// TIA Portal V18 export
VAR_GLOBAL   // PLC tag table "MemoryType"
   "PBB Off Mode Memo" AT %M200.0 : Bool;
   "PBB On Mode Memo" AT %M200.1 : Bool;
   "PBB Auto Mode Memo" AT %M200.2 : Bool;
   "Emergency Stop Button Pressed Memo" AT %M200.3 : Bool;
   "Tunnel FW Em Stop LS M Memo" AT %M200.4 : Bool;
   "Tunnel BW Em Stop LS M Memo" AT %M200.5 : Bool;
   "Start M Memo" AT %M200.6 : Bool;
   "Fuse Problem Major Memo" AT %M200.7 : Bool;
   "AutoLeveller Fault Memo" AT %M201.0 : Bool;
   "AutoLeveller Up Over Work Memo" AT %M201.1 : Bool;
   "AutoLeveller Down Over Work Memo" AT %M201.2 : Bool;
   "Driver Error Left Memo" AT %M201.3 : Bool;
   "Driver Error Right Memo" AT %M201.4 : Bool;
   "Wheel Drivers Fault Memo" AT %M201.5 : Bool;
   "SafetyShoe Siren&Info Memo" AT %M201.6 : Bool;
   "SafetyBarrier Activated Memo" AT %M201.7 : Bool;
   "Service GPU Active Memo" AT %M202.0 : Bool;
   "Fault Occurred Major Memo" AT %M202.1 : Bool;
   "Cabin Motor Driver Fault Memo" AT %M202.2 : Bool;
   "Fault Occured Minor Memo" AT %M202.3 : Bool;
   "OK Memo" AT %M202.4 : Bool;
   "FW L1 Memo" AT %M202.5 : Bool;
   "FW L2 Memo" AT %M202.6 : Bool;
   "FW L3 Memo" AT %M202.7 : Bool;
   "BW L1 Memo" AT %M203.0 : Bool;
   "BW L2 Memo" AT %M203.1 : Bool;
   "BW L3 Memo" AT %M203.2 : Bool;
   "LFT L1 Memo" AT %M203.3 : Bool;
   "LFT L2 Memo" AT %M203.4 : Bool;
   "LFT L3 Memo" AT %M203.5 : Bool;
   "RGHT L1 Memo" AT %M203.6 : Bool;
   "RGHT L2 Memo" AT %M203.7 : Bool;
   "RGHT L3 Memo" AT %M204.0 : Bool;
   "JS Mid M Memo" AT %M204.1 : Bool;
   "SafetyShoe Activated Memo" AT %M204.2 : Bool;
   "AutoLeveller Up Memo" AT %M204.3 : Bool;
   "AutoLeveller Down Memo" AT %M204.4 : Bool;
   "Down Stop Object Limit Memo" AT %M204.6 : Bool;
   "SafetyShoe Long Press Memo" AT %M204.7 : Bool;
   "SS Cable Problem Memo" AT %M205.0 : Bool;
   "AutoSafety Cross Memo" AT %M205.1 : Bool;
   "AutoLeveller FW Memo" AT %M205.2 : Bool;
   "AutoLeveller BW Memo" AT %M205.3 : Bool;
   "Autoleveler temp count Memo" AT %M205.4 : Bool;
   "Service PCA Active Memo" AT %M205.5 : Bool;
   "Service Hose Active Memo" AT %M205.6 : Bool;
   "Fuse Problem Minor Memo" AT %M205.7 : Bool;
   "Wire Up Stop PBB Memo" AT %M206.0 : Bool;
   "Slope Stop Up Memo" AT %M206.1 : Bool;
   "Wire Up Stop PBB Limit All Memo" AT %M206.2 : Bool;
   "Wire Down Stop PBB Memo" AT %M206.3 : Bool;
   "Slope Stop Down Memo" AT %M206.4 : Bool;
   "Down Stop Object Memo" AT %M206.5 : Bool;
   "Down Stop PBB All Memo" AT %M206.6 : Bool;
   "Slope Slow Down Memo" AT %M206.7 : Bool;
   "Slope Slow Up Memo" AT %M207.0 : Bool;
   "Slope Slow ALL Memo" AT %M207.1 : Bool;
   "Slow Activated Memo" AT %M207.2 : Bool;
   "Drive Slow Limit All Memo" AT %M207.3 : Bool;
   "FW Slow Limit All Memo" AT %M207.4 : Bool;
   "BW Slow Limit All Memo" AT %M207.5 : Bool;
   "FW M Memo" AT %M207.6 : Bool;
   "BW M Memo" AT %M207.7 : Bool;
   "FW-LFT Memo" AT %M208.0 : Bool;
   "FW-RGHT Memo" AT %M208.1 : Bool;
   "BW-LFT Memo" AT %M208.2 : Bool;
   "BW-RGHT Memo" AT %M208.3 : Bool;
   "Cross M Memo" AT %M208.4 : Bool;
   "FW Stop All Memo" AT %M208.5 : Bool;
   "BW Stop All Memo" AT %M208.6 : Bool;
   "LFT Stop All Memo" AT %M208.7 : Bool;
   "RGHT Stop All Memo" AT %M209.0 : Bool;
   "FW Allowed Memo" AT %M209.1 : Bool;
   "BW Allowed Memo" AT %M209.2 : Bool;
   "LFT Allowed Memo" AT %M209.3 : Bool;
   "RGHT Allowed Memo" AT %M209.4 : Bool;
   "FW-LFT Allowed Memo" AT %M209.5 : Bool;
   "FW-RGHT Allowed Memo" AT %M209.6 : Bool;
   "BW-LFT Allowed Memo" AT %M209.7 : Bool;
   "BW-RGHT Allowed Memo" AT %M210.0 : Bool;
   "Drive Angle Stop Left Memo" AT %M210.1 : Bool;
   "Drive LSW Left Stop Memo" AT %M210.2 : Bool;
   "Drive Angle Stop Right Memo" AT %M210.3 : Bool;
   "Drive LSW Right Stop Memo" AT %M210.4 : Bool;
   "Drive Slow Left Limit Memo" AT %M210.5 : Bool;
   "Drive Slow Right Limit Memo" AT %M210.6 : Bool;
   "Rotunda FW Stop LFT Memo" AT %M210.7 : Bool;
   "Rotunda BW Stop LFT Memo" AT %M211.0 : Bool;
   "Rotunda FW Stop RGHT Memo" AT %M211.1 : Bool;
   "Rotunda BW Stop RGHT Memo" AT %M211.2 : Bool;
   "Rotunda FW Stop All Memo" AT %M211.3 : Bool;
   "Rotunda BW Stop All Memo" AT %M211.4 : Bool;
   "Tunnel Laser FW Slow Limit Memo" AT %M211.5 : Bool;
   "Tunnel LSW FW Slow Memo" AT %M211.6 : Bool;
   "PhotoCell Slow Limit Memo" AT %M211.7 : Bool;
   "UltraSonic Slow Limit Memo" AT %M212.0 : Bool;
   "AirCraft Seen Anime Memo" AT %M212.1 : Bool;
   "Tunnel Laser BW Slow Limit Memo" AT %M212.2 : Bool;
   "LS BW Slow Limit Memo" AT %M212.3 : Bool;
   "Service Air Active Memo" AT %M212.4 : Bool;
   "Tunnel Laser FW Stop Limit Memo" AT %M212.5 : Bool;
   "Drive Angle LS FW Stop Memo" AT %M212.6 : Bool;
   "LS FW Stop Limit Memo" AT %M212.7 : Bool;
   "Bumper Touch LFT Stop Memo" AT %M213.0 : Bool;
   "Bumper Touch Mid Stop Memo" AT %M213.1 : Bool;
   "Bumper Touch RGTH Stop Memo" AT %M213.2 : Bool;
   "AirCraft Touch Anime Memo" AT %M213.3 : Bool;
   "Tunnel Laser BW Stop Limit Memo" AT %M213.4 : Bool;
   "LS BW Stop Limit Memo" AT %M213.5 : Bool;
   "Drive Angle LS BW Stop Memo" AT %M213.6 : Bool;
   "FW G120C Stop Memo" AT %M213.7 : Bool;
   "BW G120C Stop Memo" AT %M214.0 : Bool;
   "LFT G120C Stop Memo" AT %M214.1 : Bool;
   "Right G120C Stop Memo" AT %M214.2 : Bool;
   "FW-LFT G120C Stop Memo" AT %M214.3 : Bool;
   "FW-RGHT G120C Stop Memo" AT %M214.4 : Bool;
   "BW-LFT G120C Stop Memo" AT %M214.5 : Bool;
   "BW-RGHT G120C Stop Memo" AT %M214.6 : Bool;
   "Cab Angle Left Stop Memo" AT %M214.7 : Bool;
   "Cabin LS Left Memo" AT %M215.0 : Bool;
   "Cabin Left All Memo" AT %M215.1 : Bool;
   "Cab Angle Right Stop Memo" AT %M215.2 : Bool;
   "Cabin LS Right Memo" AT %M215.3 : Bool;
   "Cabin Right All Memo" AT %M215.4 : Bool;
   "Rotunda Stop Angle Rght Memo" AT %M215.5 : Bool;
   "Rotunda Stop Angle LFT Memo" AT %M215.6 : Bool;
   "Rotunda Slow Angle Rght Memo" AT %M215.7 : Bool;
   "Canopy BW Auto Memo" AT %M216.0 : Bool;
   "canopy ok1 Memo" AT %M216.1 : Bool;
   "canopy ok2 Memo" AT %M216.2 : Bool;
   "memo2 Memo" AT %M216.3 : Bool;
   "memo Memo" AT %M216.4 : Bool;
   "memo3 Memo" AT %M216.5 : Bool;
   "Rotunda LSW LFT Memo" AT %M216.6 : Bool;
   "Rotunda Slow Angle LFT Memo" AT %M216.7 : Bool;
   "Drive Brake Off Memo" AT %M217.0 : Bool;   // Tüm motor frenini iptal eder
   "Bumper Touch Memo" AT %M217.1 : Bool;   // Bumper orta, sag ve sol uyarılarının hepsi için
   "Canopy Touch Left Memo" AT %M217.2 : Bool;
   "Canopy Touch Right Memo" AT %M217.3 : Bool;
   "Canopy Touch Memo" AT %M217.4 : Bool;
   "Rotunda Slow Angle ALL Memo" AT %M217.6 : Bool;
   "memo4 Memo" AT %M220.0 : Bool;
   "SE ByPass Memo" AT %M220.2 : Bool;
   "Rotunda LSW Rght Memo" AT %M225.5 : Bool;
   "Slope Stop All Memo" AT %M225.6 : Bool;
   "Speed Active L1 Memo" AT %M225.7 : Bool;
   "Fast Mode Memo" AT %M226.0 : Bool;
   "Slow Mode input" AT %M226.1 : Bool;
   "Speed Active L2 Memo" AT %M226.2 : Bool;
   "Speed Active L3 Memo" AT %M226.3 : Bool;
   "R6 - Cab Warning Light & Buzzer Test Memo" AT %M226.4 : Bool;
   "Button ByPass Memo" AT %M226.5 : Bool;
   "Button Reset Memo" AT %M226.6 : Bool;
   "Tunnel Real Meter Memo" AT %MD300 : Real;
   "Drive Angle Real Meter Memo" AT %MD304 : Real;
   "Rotunda Angle Real Meter Memo" AT %MD312 : Real;
   "Height Real Memo" AT %MD332 : Real;
   "Cab Angle Real Meter Memo" AT %MD348 : Real;
   "SafetyShoe Box Status Memo" AT %M217.5 : Bool;
END_VAR
